INTERFACE ITF_LUT EXTENDS ITF_Device

END_INTERFACE

(* stored: Version 1.1.0.1, ProductVersion 3.1.4026.18
   Itf ITF_LUT: Id {6c0d6849-e396-4313-9db5-4e08f7814412} *)
